// TIA Portal V19 export
FUNCTION_BLOCK "TwoHand_FB"   // FB48, F_LAD
// stored: Access Published
   VAR_INPUT
      Enable : Bool;
      ButtonL : Bool;
      ButtonR : Bool;
      Estop : Bool;
   END_VAR
   VAR_IN_OUT
      Sts : "udt_BimanualSts";
   END_VAR
   VAR
      TWO_H_EN : TWO_H_EN;
   END_VAR
BEGIN

REGION Network 1: Two Hands LB11 - Control
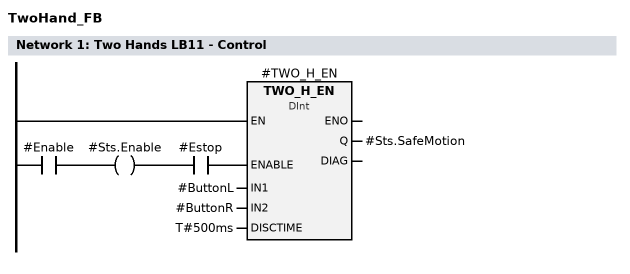
   RUNG wire#powerrail
      { S7_Templates := "codedbool_type := DInt" } #TWO_H_EN.TWO_H_EN(ENABLE := wire#w1, IN1 := #ButtonL, IN2 := #ButtonR, DISCTIME := T#500ms, Q => #Sts.SafeMotion, DIAG =>)
   END_RUNG
   RUNG wire#powerrail
      Contact( #Enable )
      Coil( #Sts.Enable )
      Contact( #Estop )
   END_RUNG wire#w1
   // the same network as SCL:
   #Sts.Enable := #Enable;
   #TWO_H_EN(ENABLE := #Enable AND #Estop,   // TWO_H_EN
             IN1 := #ButtonL,
             IN2 := #ButtonR,
             DISCTIME := T#500ms,
             Q => #Sts.SafeMotion);
END_REGION
END_FUNCTION_BLOCK
